{attribute 'qualified_only'}
{attribute 'strict'}
{attribute 'to_string'}
TYPE E_OutputLevel :
(
	SMALL := 1,
	MEDIUM := 2,
	BIG := 3,
	SUPERSTRONG := 4	
);
END_TYPE

(* stored: Version 1.1.0.1, ProductVersion 3.1.4024.12
   DUT E_OutputLevel: Id {e8345885-1238-46fd-979f-6d45b490d002} *)
